{attribute 'TcRpcEnable'}
METHOD MoveModulo : itfAxisCommand
END_METHOD

{attribute 'TcRpcEnable'}
METHOD MoveRelative : itfAxisCommand
VAR_INPUT
	Distance		: REAL;
	Velocity		: REAL;
	Acceleration	: REAL;
	Deceleration	: REAL;
//	Jerk			: REAL;
//	BufferMode		: MC_BUFFER_MODE;
	Options         : Tc3_DriveMotionControl.ST_MoveOptions;
END_VAR
VAR
	itfAxisCommand   : itfAxisCommand;
	_Command         : ST_Command;
END_VAR
MC.MoveRelative(
	Axis:= Axis, 
	Execute:= TRUE, 
	Distance:= Distance, 
	Velocity:= Velocity, 
	Acceleration:= Acceleration, 
	Deceleration:= Deceleration, 
	Options:= Options, 
	Done=> _Command.Done, 
	Busy=> _Command.Busy, 
	Active=>  _Command.Active, 
	CommandAborted=>  _Command.CommandAborted, 
	Error=> _Command.Error, 
	ErrorID=> _Command.ErrorID_Udint);
	
MC.MoveRelative(
	Axis:= Axis, 
	Execute:= FALSE);		
	
itfAxisCommand.Done 				:=  _Command.Done; //AND ActualPosition = ActualPosition + Distance;             
itfAxisCommand.Busy   				:=	_Command.Busy;
itfAxisCommand.Active 				:=	_Command.Active;
itfAxisCommand.CommandAborted		:=	_Command.CommandAborted;
itfAxisCommand.Error 				:=	_Command.Error;
itfAxisCommand.ErrorID_Udint 		:=	_Command.ErrorID_Udint;

MoveRelative := itfAxisCommand;
END_METHOD

{attribute 'TcRpcEnable'}
METHOD MoveVelocity : itfContinuousAxisCommand
VAR_INPUT
	Velocity	: REAL;
	Acceleration	: REAL;
	Deceleration	: REAL;
	Jerk	: REAL;
	Direction	: MC_Direction;
	BufferMode	: MC_BUFFER_MODE;
END_VAR
END_METHOD

{attribute 'TcRpcEnable'}
METHOD Stop : itfAxisCommand
VAR_INPUT
	Deceleration	: REAL;
	Jerk	: REAL;
END_VAR
END_METHOD

{warning 'Agregar implementación de propiedad'}
PROPERTY Error : BOOL
GET
END_GET
END_PROPERTY

{warning 'Agregar implementación de propiedad'}
PROPERTY ErrorId : WORD
GET
END_GET
END_PROPERTY

{warning 'Agregar implementación de propiedad'}
PROPERTY ErrorId_Udint_Status : UDINT
GET
END_GET
END_PROPERTY

{warning 'Agregar implementación de propiedad'}
PROPERTY IsHomed : BOOL
GET
END_GET
END_PROPERTY

{warning 'Agregar implementación de propiedad'}
PROPERTY MotionStatus : MOTION_STATUS
GET
END_GET
END_PROPERTY

{warning 'Agregar implementación de propiedad'}
PROPERTY PowerOn : BOOL
GET
PowerOn := _PowerOn;
END_GET
END_PROPERTY

{warning 'Agregar implementación de propiedad'}
PROPERTY Simulation : BOOL
GET
END_GET
END_PROPERTY

PROPERTY Status : Tc3_DriveMotionControl.MC_AxisStates
GET
VAR
	AxisStates : Tc3_DriveMotionControl.MC_AxisStates;
END_VAR
//CASE Axis.Status.MotionState OF 
//    MC_AXISSTATE_UNDEFINED : 
//         AxisStates := MC_AxisStates.MC_AXISSTATE_UNDEFINED;
//	MC_AXISSTATE_DISABLED:
//		AxisStates := MC_AxisStates.MC_AXISSTATE_DISABLED;
//	MC_AXISSTATE_STANDSTILL:
//		AxisStates := MC_AxisStates.MC_AXISSTATE_STANDSTILL;
//	MC_AXISSTATE_ERRORSTOP:		
//		AxisStates := MC_AxisStates.MC_AXISSTATE_ERRORSTOP;
//	MC_AXISSTATE_STOPPING:			
//		AxisStates := MC_AxisStates.MC_AXISSTATE_STOPPING;
//	MC_AXISSTATE_HOMING:			
//		AxisStates := MC_AxisStates.MC_AXISSTATE_HOMING;
//	MC_AXISSTATE_DISCRETEMOTION:			
//		AxisStates := MC_AxisStates.MC_AXISSTATE_DISCRETEMOTION;
//	MC_AXISSTATE_CONTINOUSMOTION:			
//		AxisStates := MC_AxisStates.MC_AXISSTATE_CONTINOUSMOTION;
////	MC_AXISSTATE_SYNCHRONIZEDMOTION:			
////		AxisStates := MC_AxisStates.MC_AXISSTATE_SYNCHRONIZEDMOTION;
//END_CASE;

//Status := AxisStates;

Status := Axis.Status.MotionState;
END_GET
END_PROPERTY

{warning 'Agregar implementación de método'}
METHOD AbortTrigger : itfCommand
END_METHOD

{warning 'Agregar implementación de método'}
METHOD TouchProbe : itfCommand
END_METHOD

END_FUNCTION_BLOCK

// TwinCAT Library Template/VendorImplementation/TcAxis_Base
FUNCTION_BLOCK ABSTRACT TcAxis_Base IMPLEMENTS itfAxis_Tc3_DriveMotionControl
//VAR_INPUT
//END_VAR
//VAR_OUTPUT
//END_VAR
//VAR
//END_VAR

{warning 'Agregar implementación de propiedad'}
PROPERTY ActualPosition : REAL
GET
END_GET
END_PROPERTY

{warning 'Agregar implementación de propiedad'}
PROPERTY ActualVelocity : REAL
GET
END_GET
END_PROPERTY

{attribute 'TcRpcEnable'}
{warning 'Agregar implementación de método'}
METHOD ABSTRACT Power : itfCommand
VAR_INPUT
//	Enable	: BOOL;
//	EnablePositive	: BOOL;
//	EnableNegative	: BOOL;
END_VAR
END_METHOD

{attribute 'TcRpcEnable'}
{warning 'Agregar implementación de método'}
METHOD Reset : itfCommand
END_METHOD

{warning 'Agregar implementación de método'}
METHOD SetPosition : itfCommand
VAR_INPUT
	Position	: REAL;
	Relative	: BOOL;
	(*	ExecutionMode	: MC_ExecutionMode;*)
	ExecutionMode	: Tc2_MC2.ST_SetPositionOptions;
END_VAR
END_METHOD

{warning 'Agregar implementación de método'}
METHOD Halt : itfAxisCommand
VAR_INPUT
	Deceleration	: REAL;
	Jerk	: REAL;
	BufferMode	: MC_BUFFER_MODE;
END_VAR
END_METHOD

{warning 'Agregar implementación de método'}
METHOD Home : itfAxisCommand
VAR_INPUT
	Position	: REAL;
	Velocity	: REAL;
	EndVelocity	: REAL;
	Acceleration	: REAL;
	Deceleration	: REAL;
	Jerk	: REAL;
	Direction	: MC_Direction;
	HomingMode	: INT;
	BufferMode	: MC_BUFFER_MODE;
END_VAR
END_METHOD

{warning 'Agregar implementación de método'}
METHOD Jog : itfAxisCommand
VAR_INPUT
	JogForward	: BOOL;
	JogBackwards	: BOOL;
	Mode	: Tc2_MC2.E_JogMode;
	Position	: LREAL;
	Velocity	: LREAL;
	Acceleration	: LREAL;
	Deceleration	: LREAL;
	Jerk	: LREAL;
END_VAR
END_METHOD

{attribute 'TcRpcEnable'}
{warning 'Agregar implementación de método'}
METHOD ABSTRACT MoveAbsolute : itfAxisCommand
VAR_INPUT
//	Position	: REAL;
//	Velocity	: REAL;
//	Acceleration	: REAL;
//	Deceleration	: REAL;
//	Jerk	: REAL;
//	Direction	: MC_Direction;
//	BufferMode	: MC_BUFFER_MODE;
END_VAR
END_METHOD

{warning 'Agregar implementación de método'}
METHOD MoveModulo : itfAxisCommand
END_METHOD

{attribute 'TcRpcEnable'}
{warning 'Agregar implementación de método'}
METHOD MoveRelative : itfAxisCommand
VAR_INPUT
	Distance	: REAL;
	Velocity	: REAL;
	Acceleration	: REAL;
	Deceleration	: REAL;
	Jerk	: REAL;
	BufferMode	: MC_BUFFER_MODE;
END_VAR
END_METHOD

{warning 'Agregar implementación de método'}
METHOD MoveVelocity : itfContinuousAxisCommand
VAR_INPUT
	Velocity	: REAL;
	Acceleration	: REAL;
	Deceleration	: REAL;
	Jerk	: REAL;
	Direction	: MC_Direction;
	BufferMode	: MC_BUFFER_MODE;
END_VAR
END_METHOD

{warning 'Agregar implementación de método'}
METHOD Stop : itfAxisCommand
VAR_INPUT
	Deceleration	: REAL;
	Jerk	: REAL;
END_VAR
END_METHOD

{warning 'Agregar implementación de propiedad'}
PROPERTY Error : BOOL
GET
END_GET
END_PROPERTY

{warning 'Agregar implementación de propiedad'}
PROPERTY ErrorId : WORD
GET
END_GET
END_PROPERTY

{warning 'Agregar implementación de propiedad'}
PROPERTY ErrorId_Udint_Status : UDINT
GET
END_GET
END_PROPERTY

{warning 'Agregar implementación de propiedad'}
PROPERTY IsHomed : BOOL
GET
END_GET
END_PROPERTY

{warning 'Agregar implementación de propiedad'}
PROPERTY MotionStatus : MOTION_STATUS
GET
END_GET
END_PROPERTY

{warning 'Agregar implementación de propiedad'}
PROPERTY PowerOn : BOOL
GET
END_GET
END_PROPERTY

{warning 'Agregar implementación de propiedad'}
PROPERTY Simulation : BOOL
GET
END_GET
END_PROPERTY

PROPERTY Status : MC_AxisStates
GET
END_GET
END_PROPERTY

{warning 'Agregar implementación de método'}
METHOD AbortTrigger : itfCommand
END_METHOD

{warning 'Agregar implementación de método'}
METHOD TouchProbe : itfCommand
END_METHOD

END_FUNCTION_BLOCK

// TwinCAT Library Template/Part1Definition/Interfaces/itfAxis_Tc3_DriveMotionControl
INTERFACE itfAxis_Tc3_DriveMotionControl

{warning 'add property implementation'}
PROPERTY ActualPosition : REAL
GET
END_GET
END_PROPERTY

{warning 'add property implementation'}
PROPERTY ActualVelocity : REAL
GET
END_GET
END_PROPERTY

{attribute 'TcRpcEnable'}
//METHOD ABSTRACT Power	: itfCommand
METHOD Power	: itfCommand
VAR_INPUT
	Enable				: BOOL;
//	EnablePositive		: BOOL;
//	EnableNegative		: BOOL;
END_VAR
END_METHOD

{attribute 'TcRpcEnable'}
METHOD Reset : itfCommand
END_METHOD

{attribute 'TcRpcEnable'}
METHOD SetPosition 	: itfCommand
VAR_INPUT
	Position		: REAL;
	Relative		: BOOL;
//	ExecutionMode	: MC_ExecutionMode;
	ExecutionMode	: Tc2_MC2.ST_SetPositionOptions;
END_VAR
END_METHOD

{attribute 'TcRpcEnable'}
METHOD Halt 		: itfAxisCommand
VAR_INPUT
	Deceleration	: REAL;
	Jerk			: REAL;
	BufferMode		: MC_BUFFER_MODE;
END_VAR
END_METHOD

{attribute 'TcRpcEnable'}
METHOD Home 		: itfAxisCommand
VAR_INPUT
	Position		: REAL;
	Velocity		: REAL;
	EndVelocity		: REAL;
	Acceleration	: REAL;
	Deceleration	: REAL;
	Jerk			: REAL;
	Direction		: MC_Direction;
	HomingMode		: INT;
	BufferMode		: MC_BUFFER_MODE;
END_VAR
END_METHOD

{attribute 'TcRpcEnable'}
METHOD Jog 			: itfAxisCommand
VAR_INPUT
    JogForward 		: BOOL;
    JogBackwards 	: BOOL;
    Mode     		: Tc2_MC2.E_JogMode;
    Position        : LREAL;
    Velocity        : LREAL;
    Acceleration 	: LREAL;
    Deceleration 	: LREAL;
    Jerk     		: LREAL;
END_VAR
END_METHOD

{attribute 'TcRpcEnable'}
METHOD MoveAbsolute : itfAxisCommand
//METHOD ABSTRACT MoveAbsolute : itfAxisCommand
VAR_INPUT
	Position		: REAL;
	Velocity		: REAL;
	Acceleration	: REAL;
	Deceleration	: REAL;
//	Jerk			: REAL;
//	Direction		: MC_Direction;
//	BufferMode		: MC_BUFFER_MODE;
	Options         : Tc3_DriveMotionControl.ST_MoveOptions;
END_VAR
END_METHOD

{attribute 'TcRpcEnable'}
METHOD MoveModulo : itfAxisCommand
VAR_INPUT
END_VAR
END_METHOD

{attribute 'TcRpcEnable'}
METHOD MoveRelative : itfAxisCommand
VAR_INPUT
	Distance		: REAL;
	Velocity		: REAL;
	Acceleration	: REAL;
	Deceleration	: REAL;
//	Jerk			: REAL;
//	BufferMode		: MC_BUFFER_MODE;
	Options         : Tc3_DriveMotionControl.ST_MoveOptions;
END_VAR
END_METHOD

{attribute 'TcRpcEnable'}
METHOD MoveVelocity : itfContinuousAxisCommand
VAR_INPUT
	Velocity		: REAL;
	Acceleration	: REAL;
	Deceleration	: REAL;
	Jerk			: REAL;
	Direction		: MC_Direction;
	BufferMode		: MC_BUFFER_MODE;
END_VAR
END_METHOD

{attribute 'TcRpcEnable'}
METHOD Stop 		: itfAxisCommand
VAR_INPUT
	Deceleration	: REAL;
	Jerk			: REAL;
END_VAR
END_METHOD

PROPERTY Error : BOOL
GET
END_GET
END_PROPERTY

{warning 'add property implementation'}
PROPERTY ErrorId : WORD
GET
END_GET
END_PROPERTY

PROPERTY ErrorId_Udint_Status : UDINT
GET
END_GET
END_PROPERTY


PROPERTY IsHomed : BOOL
GET
END_GET
END_PROPERTY

{warning 'add property implementation'}
PROPERTY MotionStatus : MOTION_STATUS
GET
END_GET
END_PROPERTY

{attribute ‘monitoring’ := ‘call’}
PROPERTY PowerOn : BOOL
GET
END_GET
END_PROPERTY

{warning 'add property implementation'}
PROPERTY Simulation : BOOL
GET
END_GET
END_PROPERTY

PROPERTY Status : Tc3_DriveMotionControl.MC_AxisStates
GET
END_GET
END_PROPERTY

METHOD AbortTrigger : itfCommand
VAR_INPUT
END_VAR
END_METHOD

METHOD TouchProbe : itfCommand
VAR_INPUT
END_VAR
END_METHOD

END_INTERFACE

// Examples/_MAIN_Examples
PROGRAM _MAIN_Examples
VAR
//	fbAxis_X1 				: TcAxis_Tc2_MC2;
			
//	fbSum : FB_Sum;
END_VAR

//Examples Tc2_MC2:
WareHousingExample_Tc2_MC2();
//LabelingExample();
//CamGearExample();

//Examples Tc3_DriveMotionControl:
WareHousingExample_Tc3_DriveMotionControl();

END_PROGRAM

// Examples/LabelingExample
PROGRAM LabelingExample
VAR
	AXIS_REF_LabelDrive			: TC2_MC2.AXIS_REF;
	AXIS_REF_Conveyor 			: TC2_MC2.AXIS_REF;

	// Hardware definitions
	LabelDrive 			: TcAxis_Tc2_MC2;
	Conveyor 			: TcAxis_Tc2_MC2;
	LabelLength 		: REAL := 100;
	SensorDistance 		: REAL := 10;
	Velocity 			: REAL := 5;
	ProductDetection 	: BOOL := FALSE;
	DelayTimer 			: TON;
	
	// States
	ConveyorState 		: INT := 0;
	LabelDriveState 	: INT := 0;
	
	// Control
	Start 				: BOOL := FALSE;
	
	// Commands
	ConveyorMove 		: itfCommand;
	LabelDriveMove 		: itfCommand;
END_VAR


LabelDrive(Axis:= AXIS_REF_LabelDrive);
Conveyor(Axis:= AXIS_REF_Conveyor);

// Run the timer. As it is a classic FB it should be called every cycle
DelayTimer(IN:=ProductDetection, PT:= INT_TO_TIME(REAL_TO_INT(SensorDistance * 1000 / Velocity)));

CASE ConveyorState OF
	0: // Disabled
		IF Start THEN
			ConveyorState := ConveyorState + 1;
		END_IF
		
	1: // Power On
		Conveyor.Power(Enable:=TRUE, EnablePositive:=TRUE, EnableNegative:=TRUE);
		//IF Conveyor.Status = AXIS_STATUS.Standstill THEN
	  IF Conveyor.Status = Tc2_MC2.MC_AXISSTATE_STANDSTILL THEN
			ConveyorState := ConveyorState + 1;
		END_IF
		
	2: // Wait for LabelDrive 
		//IF LabelDrive.Status = AXIS_STATUS.Standstill THEN
		IF LabelDrive.Status =  Tc2_MC2.MC_AXISSTATE_STANDSTILL THEN
			ConveyorMove := Conveyor.MoveVelocity(Velocity:=Velocity, Acceleration:=0, Deceleration:=0, Jerk:=0, Direction:=MC_Direction.mcPositiveDirection, BufferMode:=MC_BUFFER_MODE.mcAborting);
			ConveyorState := ConveyorState + 1;
		END_IF
		
	3: // Moving
		IF NOT Start THEN
			ConveyorMove := Conveyor.Halt(Deceleration:=0, Jerk:=0, BufferMode:=MC_BUFFER_MODE.mcAborting);
			ConveyorState := ConveyorState + 1;
		END_IF
		
	4: // Stopping
		IF ConveyorMove.Done THEN
			ConveyorState := ConveyorState + 1;
		END_IF
		
	5: // Power off
		Conveyor.Power(Enable:=FALSE, EnablePositive:=FALSE, EnableNegative:=FALSE);
		IF Conveyor.Status = AXIS_STATUS.Disabled THEN
			ConveyorState := 0;
		END_IF
END_CASE

CASE LabelDriveState OF
	0: // Disabled
		IF Start THEN
			LabelDriveState := LabelDriveState + 1;
		END_IF
		
	1: // Power On
		LabelDrive.Power(Enable:=TRUE, EnablePositive:=TRUE, EnableNegative:=TRUE);
		//IF LabelDrive.Status = AXIS_STATUS.Standstill THEN
		IF LabelDrive.Status = Tc2_MC2.MC_AXISSTATE_STANDSTILL THEN
			LabelDriveState := LabelDriveState + 1;
		END_IF
		
	2: // Wait for Conveyor 
		//IF Conveyor.Status = AXIS_STATUS.Standstill THEN
		IF Conveyor.Status = Tc2_MC2.MC_AXISSTATE_STANDSTILL THEN
			LabelDriveState := LabelDriveState + 1;
		END_IF
						
	3: // Wait for product
		IF NOT Start THEN
			LabelDriveState := 5;
		END_IF
		IF DelayTimer.Q THEN
			LabelDriveMove := LabelDrive.MoveRelative(Distance:=LabelLength, Velocity:=Velocity, Acceleration:=0, Deceleration:=0, Jerk:=0, BufferMode:=MC_BUFFER_MODE.mcAborting);
			LabelDriveState := LabelDriveState + 1;
		END_IF
		
	4: // Wait for label to be transfered
		IF LabelDriveMove.Done AND NOT DelayTimer.Q THEN
			LabelDriveState := 3;
		END_IF
		
	5: // Power off
		Conveyor.Power(Enable:=FALSE, EnablePositive:=FALSE, EnableNegative:=FALSE);
		IF Conveyor.Status = AXIS_STATUS.Disabled THEN
			LabelDriveState := 0;
		END_IF
	
END_CASE

END_PROGRAM

// Examples/CamGearExample
PROGRAM CamGearExample
VAR
	// Hardware definitions
	TcMasterDrive 	: TcAxis_Tc2_MC2;
	TcCamDrive 		: TcAxis_Tc2_MC2;
	TcGearDrive 	: TcAxis_Tc2_MC2;
	
	
	MasterDrive 	: itfAxis_Tc2_MC2;
	CamDrive 		: itfAxis_Tc2_MC2;
	GearDrive 		: itfAxis_Tc2_MC2;
	Table 			: TcCamTable;
	TableData 		: MC_CAM_REF;
	Velocity 		: REAL := 5;
	
	// States
	MasterState 	: INT := 0;
	CamState 		: INT := 0;
	GearState 		: INT := 0;
	
	// Control
	Start 			: BOOL := FALSE;
	
	// Commands
	MasterMove 		: itfCommand;
	TableSet 		: itfCommand;
	CamMove 		: itfSynchronizedAxisCommand;
	GearMove 		: itfSynchronizedAxisCommand;
END_VAR


MasterDrive:= TcMasterDrive;
CamDrive := TcCamDrive;
GearDrive := TcGearDrive;

CASE MasterState OF
	0: // Disabled
		IF Start THEN
			MasterState := MasterState + 1;
		END_IF
		
	1: // Power On
		MasterDrive.Power(Enable:=TRUE, EnablePositive:=TRUE, EnableNegative:=TRUE);
		IF MasterDrive.Status = AXIS_STATUS.Standstill THEN
			MasterState := MasterState + 1;
		END_IF
		
	2: // Wait for other drives 
		IF CamMove.InSync AND GearMove.InSync THEN
			MasterMove := MasterDrive.MoveVelocity(Velocity:=Velocity, Acceleration:=0, Deceleration:=0, Jerk:=0, Direction:=MC_Direction.mcPositiveDirection, BufferMode:=MC_BUFFER_MODE.mcAborting);
			MasterState := MasterState + 1;
		END_IF
		
	3: // Moving
		IF NOT Start THEN
			MasterMove:= MasterDrive.Halt(Deceleration:=0, Jerk:=0, BufferMode:=MC_BUFFER_MODE.mcAborting);
			MasterState := MasterState + 1;
		END_IF
		
	4: // Stopping
		IF NOT MasterMove.Done THEN
			MasterState := MasterState + 1;
		END_IF
		
	5: // Power off
		MasterDrive.Power(Enable:=FALSE, EnablePositive:=FALSE, EnableNegative:=FALSE);
		IF MasterDrive.Status = AXIS_STATUS.Disabled THEN
			MasterState := 0;
		END_IF
END_CASE

CASE CamState OF
	0: // Disabled
		IF Start THEN
			CamState := CamState + 1;
		END_IF
		
	1: // Power On
		CamDrive.Power(Enable:=TRUE, EnablePositive:=TRUE, EnableNegative:=TRUE);
		IF CamDrive.Status = AXIS_STATUS.Standstill AND MasterDrive.Status = AXIS_STATUS.Standstill THEN
			TableSet := Table.Select(CamTable:=TableData, Periodic:=TRUE, MasterAbsolute:=TRUE, SlaveAbsolute:=TRUE);
			CamState := CamState + 1;
		END_IF
		
	2: // Set CAM Table
		IF TableSet.Done THEN
			CamMove := CamDrive.CamIn(Master:=MasterDrive, MasterOffset:=0, SlaveOffset:=0, MasterScaling:=1, SlaveScaling:=1, MasterStartDistance:=0, MasterSyncPosition:=0, 
				StartMode:=MC_StartMode.mcRelative, MasterValueSource:=MC_Source.mcSetValue,CamTable:=Table, BufferMode:=MC_BUFFER_MODE.mcAborting);
			CamState := CamState + 1;
		END_IF
		
	3: // Synchronized
		IF NOT Start THEN
			CamDrive.Release();
			CamState := CamState + 1;
		END_IF
		
	4: // Power off
		CamDrive.Power(Enable:=FALSE, EnablePositive:=FALSE, EnableNegative:=FALSE);
		IF CamDrive.Status = AXIS_STATUS.Disabled THEN
			CamState := 0;
		END_IF
END_CASE

CASE GearState OF
	0: // Disabled
		IF Start THEN
			GearState := GearState + 1;
		END_IF
		
	1: // Power On
		GearDrive.Power(Enable:=TRUE, EnablePositive:=TRUE, EnableNegative:=TRUE);
		IF GearDrive.Status = AXIS_STATUS.Standstill AND MasterDrive.Status = AXIS_STATUS.Standstill THEN
			GearMove := GearDrive.GearIn(Master:=MasterDrive, Ratio:=2, MasterValueSource:=MC_Source.mcSetValue,Acceleration:=0, Deceleration:=0, Jerk:=0, BufferMode:=MC_BUFFER_MODE.mcAborting);
			GearState := GearState + 1;
		END_IF
		
	2: // Synchronized
		IF NOT Start THEN
			GearDrive.Release();
			GearState := GearState + 1;
		END_IF
		
	3: // Power off
		GearDrive.Power(Enable:=FALSE, EnablePositive:=FALSE, EnableNegative:=FALSE);
		IF GearDrive.Status = AXIS_STATUS.Disabled THEN
			GearState := 0;
		END_IF
END_CASE

END_PROGRAM

// TwinCAT Library Template/VendorImplementation/TcCamTable
FUNCTION_BLOCK TcCamTable IMPLEMENTS itfCamTable
VAR_INPUT
END_VAR
VAR_OUTPUT
END_VAR
VAR
END_VAR

{warning 'add method implementation '}
METHOD Select 		: itfCommand
VAR_INPUT	
	Periodic		: BOOL;
	MasterAbsolute	: BOOL;
	SlaveAbsolute	: BOOL;
	CamTable		: MC_CAM_REF;
END_VAR
VAR
	
END_VAR
END_METHOD

END_FUNCTION_BLOCK

// Project Information/F_GetCompany
// This function has been automatically generated from the project information.
{attribute 'signature_flag' := '1073741824'}
{attribute 'TcGenerated'}
{attribute 'no-analysis'}
FUNCTION F_GetCompany : WSTRING
VAR_INPUT
	
END_VAR

F_GetCompany := "TcMotion";

END_FUNCTION

// Project Information/F_GetTitle
// This function has been automatically generated from the project information.
{attribute 'signature_flag' := '1073741824'}
{attribute 'TcGenerated'}
{attribute 'no-analysis'}
FUNCTION F_GetTitle : WSTRING
VAR_INPUT
	
END_VAR

F_GetTitle := "TcMotion_Component";

END_FUNCTION

// Project Information/F_GetVersion
// This function has been automatically generated from the project information.
{attribute 'signature_flag' := '1073741824'}
{attribute 'TcGenerated'}
{attribute 'no-analysis'}
FUNCTION F_GetVersion : ST_LibVersion
VAR_INPUT
	
END_VAR

F_GetVersion.iMajor := 1;
F_GetVersion.iMinor := 0;
F_GetVersion.iBuild := 0;
F_GetVersion.iRevision := 8;
F_GetVersion.sVersion := '1.0.0.8';
F_GetVersion.nFlags := 0;

END_FUNCTION

// TwinCAT Library Template/Part1Definition/Interfaces/itfAxis_Tc2_MC2_Camming
INTERFACE itfAxis_Tc2_MC2_Camming

(*
!!!! It would have to be another library with this new extension for the Axis, because if not in TwinCAT this new license is added:
!!!! TF5050 TC3 NC Camming !!!!!!*)

{attribute 'TcRpcEnable'}
METHOD CamIn 			: itfSynchronizedAxisCommand
VAR_INPUT
//	Master				: itfAxis;
	Master				: Tc2_MC2.AXIS_REF;
	Slave				: Tc2_MC2.AXIS_REF;	
	MasterOffset		: REAL;
	SlaveOffset			: REAL;
	MasterScaling		: REAL;
	SlaveScaling		: REAL;
	MasterStartDistance	: REAL;
	MasterSyncPosition	: REAL;
	StartMode			: MC_StartMode;
	MasterValueSource	: MC_Source;
//	CamTable			: itfCamTable;
	CamTableID			: Tc2_MC2_Camming.MC_CAM_ID;
	BufferMode			: MC_BUFFER_MODE;
END_VAR
END_METHOD

{attribute 'TcRpcEnable'}
METHOD CamOut : : itfSynchronizedAxisCommand
VAR_INPUT
END_VAR
END_METHOD

{attribute 'TcRpcEnable'}
METHOD CamScaling : itfSynchronizedAxisCommand
VAR_INPUT
END_VAR
END_METHOD

{attribute 'TcRpcEnable'}
METHOD CamTableSelect  : itfSynchronizedAxisCommand
VAR_INPUT
END_VAR
END_METHOD

{attribute 'TcRpcEnable'}
METHOD ReadMotionFunction : itfSynchronizedAxisCommand
VAR_INPUT
END_VAR
END_METHOD

{attribute 'TcRpcEnable'}
METHOD ReadMotionFunctionPoint : itfSynchronizedAxisCommand
VAR_INPUT
END_VAR
END_METHOD

{attribute 'TcRpcEnable'}
METHOD ReadMotionFunctionValues : itfSynchronizedAxisCommand
VAR_INPUT
END_VAR
END_METHOD

{attribute 'TcRpcEnable'}
METHOD SetCamOnlineChangeMode : itfSynchronizedAxisCommand
VAR_INPUT
END_VAR
END_METHOD

{attribute 'TcRpcEnable'}
METHOD WriteMotionFunction : itfSynchronizedAxisCommand
VAR_INPUT
END_VAR
END_METHOD

{attribute 'TcRpcEnable'}
METHOD WriteMotionFunctionPoint : itfSynchronizedAxisCommand
VAR_INPUT
END_VAR
END_METHOD

{attribute 'TcRpcEnable'}
METHOD CamAdd : itfSynchronizedAxisCommand
VAR_INPUT
END_VAR
END_METHOD

{attribute 'TcRpcEnable'}
METHOD CamExchange : itfSynchronizedAxisCommand
VAR_INPUT
END_VAR
END_METHOD

{attribute 'TcRpcEnable'}
METHOD CamIn_V2 : itfSynchronizedAxisCommand
VAR_INPUT
END_VAR
END_METHOD

{attribute 'TcRpcEnable'}
METHOD CamRemove : itfSynchronizedAxisCommand
VAR_INPUT
END_VAR
END_METHOD

{attribute 'TcRpcEnable'}
METHOD CamScaling_V2 : itfSynchronizedAxisCommand
VAR_INPUT
END_VAR
END_METHOD

{attribute 'TcRpcEnable'}
METHOD CamInfo : itfSynchronizedAxisCommand
VAR_INPUT
END_VAR
END_METHOD

{attribute 'TcRpcEnable'}
METHOD CamInfo_V2 : itfSynchronizedAxisCommand
VAR_INPUT
END_VAR
END_METHOD

{attribute 'TcRpcEnable'}
METHOD ReadCamTableCharacteristics : itfSynchronizedAxisCommand
VAR_INPUT
END_VAR
END_METHOD

{attribute 'TcRpcEnable'}
METHOD ReadCamTableMasterPosition : itfSynchronizedAxisCommand
VAR_INPUT
END_VAR
END_METHOD

{attribute 'TcRpcEnable'}
METHOD ReadCamTableSlaveDynamics : itfSynchronizedAxisCommand
VAR_INPUT
END_VAR
END_METHOD

END_INTERFACE

// TwinCAT Library Template/Part1Definition/Interfaces/itfAxis_Tc2_MC2_FlyingSaw
INTERFACE itfAxis_Tc2_MC2_FlyingSaw

(*
!!!! It would have to be another library with this new extension for the Axis, because if not in TwinCAT this new license is added:
!!!! TF5055 TC3 NC Flying Saw !!!!!!*)

{attribute 'TcRpcEnable'}
METHOD GearInPos 		: itfSynchronizedAxisCommand
VAR_INPUT
//	Master				: itfAxis;
	Master				: Tc2_MC2.AXIS_REF;
	Slave				: Tc2_MC2.AXIS_REF;			
	RatioNumerator		: REAL;
	RatioDenominator	: REAL;
	MasterValueSource	: MC_SOURCE;
	MasterSyncPosition	: REAL;
	SlaveSyncPosition	: REAL;
	SyncMode			: MC_SYNC_MODE;
	MasterStartDistance	: REAL;
	Velocity			: REAL;
	Acceleration		: REAL;
	Deceleration		: REAL;
	Jerk				: REAL;
	BufferMode			: MC_BUFFER_MODE;
END_VAR
END_METHOD

{attribute 'TcRpcEnable'}
METHOD GearInVelo 		: itfSynchronizedAxisCommand
VAR_INPUT
//	Master				: itfAxis;
	Master				: Tc2_MC2.AXIS_REF;
	Slave				: Tc2_MC2.AXIS_REF;			
	RatioNumerator		: REAL;
	RatioDenominator	: REAL;
	MasterValueSource	: MC_SOURCE;
	MasterSyncPosition	: REAL;
	SlaveSyncPosition	: REAL;
	SyncMode			: MC_SYNC_MODE;
	MasterStartDistance	: REAL;
	Velocity			: REAL;
	Acceleration		: REAL;
	Deceleration		: REAL;
	Jerk				: REAL;
	BufferMode			: MC_BUFFER_MODE;
END_VAR
END_METHOD

{attribute 'TcRpcEnable'}
METHOD ReadFlyingSawCharacteristics : itfSynchronizedAxisCommand
VAR_INPUT
END_VAR
END_METHOD

END_INTERFACE

// TwinCAT Library Template/VendorImplementation/TcAxis_Tc2_MC2_Camming
FUNCTION_BLOCK TcAxis_Tc2_MC2_Camming EXTENDS TcAxis_Tc2_MC2 IMPLEMENTS itfAxis_Tc2_MC2_Camming
VAR_INPUT
END_VAR
VAR_OUTPUT
END_VAR
VAR
END_VAR

{error 'Agregar implementación de método o eliminar método para utilizar la implementación básica.'}
(*
!!!! It would have to be another library with this new extension for the Axis, because if not in TwinCAT this new license is added:
!!!! TF5050 TC3 NC Camming !!!!!!*)
METHOD CamIn : itfSynchronizedAxisCommand
VAR_INPUT
	(*	Master				: itfAxis;*)
	Master	: Tc2_MC2.AXIS_REF;
	Slave	: Tc2_MC2.AXIS_REF;
	MasterOffset	: REAL;
	SlaveOffset	: REAL;
	MasterScaling	: REAL;
	SlaveScaling	: REAL;
	MasterStartDistance	: REAL;
	MasterSyncPosition	: REAL;
	StartMode	: MC_StartMode;
	MasterValueSource	: MC_Source;
	(*	CamTable			: itfCamTable;*)
	CamTableID	: Tc2_MC2_Camming.MC_CAM_ID;
	BufferMode	: MC_BUFFER_MODE;
END_VAR

VAR
	fbCamIn			 	: Tc2_MC2_Camming.MC_CamIn;	
END_VAR
(*
!!!! It would have to be another library with this new extension for the Axis, because if not in TwinCAT this new license is added:
!!!! TF5050 TC3 NC Camming !!!!!!*)

fbCamIn(
	Master:= Master, 
	Slave:= Slave, 
	Execute:= TRUE, 
	MasterOffset:= MasterOffset, 
	SlaveOffset:= SlaveOffset, 
	MasterScaling:= MasterScaling, 
	SlaveScaling:= SlaveScaling, 
	StartMode:= StartMode, 
	CamTableID:= CamTableID, //CamTable, 
	BufferMode:= , //BufferMode, 
	Options:= , 
	InSync=> , 
	Busy=> , 
	Active=> , 
	CommandAborted=> , 
	Error=> , 
	ErrorID=> );

count_delete  := count_delete + 1;
END_METHOD

END_FUNCTION_BLOCK

// TwinCAT Library Template/VendorImplementation/TcAxis_Tc2_MC2_FlyingSaw
FUNCTION_BLOCK TcAxis_Tc2_MC2_FlyingSaw EXTENDS TcAxis_Tc2_MC2 IMPLEMENTS itfAxis_Tc2_MC2_FlyingSaw
VAR_INPUT
END_VAR
VAR_OUTPUT
END_VAR
VAR
END_VAR

{error 'Agregar implementación de método o eliminar método para utilizar la implementación básica.'}
(*
!!!! It would have to be another library with this new extension for the Axis, because if not in TwinCAT this new license is added:
!!!! TF5055 TC3 NC Flying Saw !!!!!!*)
METHOD GearInPos : itfSynchronizedAxisCommand
VAR_INPUT
	(*	Master				: itfAxis;*)
	Master	: Tc2_MC2.AXIS_REF;
	Slave	: Tc2_MC2.AXIS_REF;
	RatioNumerator	: REAL;
	RatioDenominator	: REAL;
	MasterValueSource	: MC_SOURCE;
	MasterSyncPosition	: REAL;
	SlaveSyncPosition	: REAL;
	SyncMode	: MC_SYNC_MODE;
	MasterStartDistance	: REAL;
	Velocity	: REAL;
	Acceleration	: REAL;
	Deceleration	: REAL;
	Jerk	: REAL;
	BufferMode	: MC_BUFFER_MODE;
END_VAR

VAR
	fbGearInPos			: Tc2_MC2_FlyingSaw.MC_GearInPos;	
END_VAR
(*
!!!! It would have to be another library with this new extension for the Axis, because if not in TwinCAT this new license is added:
!!!! TF5055 TC3 NC Flying Saw !!!!!!*)

fbGearInPos(
	Master:= Master, 
	Slave:= Slave, 
	Execute:= , 
	RatioNumerator:= , 
	RatioDenominator:= , 
	MasterSyncPosition:= , 
	SlaveSyncPosition:= , 
	SyncMode:= , 
	MasterStartDistance:= , 
	Velocity:= , 
	Acceleration:= , 
	Deceleration:= , 
	Jerk:= , 
	BufferMode:= , 
	Options:= , 
	StartSync=> , 
	InSync=> , 
	Busy=> , 
	Active=> , 
	CommandAborted=> , 
	Error=> , 
	ErrorID=> );


count_delete  := count_delete + 1;
END_METHOD

END_FUNCTION_BLOCK

// TwinCAT Library Template/VendorImplementation/TcContinuousAxisCommand
FUNCTION_BLOCK TcContinuousAxisCommand IMPLEMENTS itfContinuousAxisCommand
VAR_INPUT
END_VAR
VAR_OUTPUT
END_VAR
VAR
END_VAR

{warning 'add method implementation '}
METHOD Abort : MC_Error
END_METHOD

{warning 'add property implementation'}
PROPERTY Active : BOOL
GET
END_GET
END_PROPERTY

{warning 'add property implementation'}
PROPERTY Busy : BOOL
GET
END_GET
END_PROPERTY

{warning 'add property implementation'}
PROPERTY Command : MC_COMMAND_REF
GET
END_GET
END_PROPERTY

{warning 'add property implementation'}
PROPERTY CommandAborted : BOOL
GET
END_GET
END_PROPERTY

{warning 'add property implementation'}
PROPERTY Done : BOOL
GET
END_GET
END_PROPERTY

{warning 'add property implementation'}
PROPERTY Error : BOOL
GET
END_GET
END_PROPERTY

{warning 'add property implementation'}
PROPERTY ErrorId : MC_Error
GET
END_GET
END_PROPERTY

{warning 'add property implementation'}
PROPERTY InVelocity : BOOL
GET
END_GET
END_PROPERTY

{warning 'add method implementation '}
METHOD Update 		: MC_Error
VAR_INPUT
	Position		: REAL;
	Velocity		: REAL;
	EndVelocity		: REAL;
	Acceleration	: REAL;
	Deceleration	: REAL;
	Jerk			: REAL;
END_VAR
END_METHOD

{warning 'add method implementation '}
METHOD Wait 		: MC_Error (* This method only makes sense in the IEC 61499 environment*)
VAR_INPUT
	Timeout			: TIME;
	AbortOnTimeout	: BOOL;
END_VAR
END_METHOD

END_FUNCTION_BLOCK

// TwinCAT Library Template/VendorImplementation/TcSynchronizedAxisCommand
FUNCTION_BLOCK TcSynchronizedAxisCommand IMPLEMENTS itfSynchronizedAxisCommand
VAR_INPUT
END_VAR
VAR_OUTPUT
END_VAR
VAR
END_VAR

{warning 'add method implementation '}
METHOD Abort : MC_Error
END_METHOD

{warning 'add property implementation'}
PROPERTY Active : BOOL
GET
END_GET
END_PROPERTY

{warning 'add property implementation'}
PROPERTY Busy : BOOL
GET
END_GET
END_PROPERTY

{warning 'add property implementation'}
PROPERTY Command : MC_COMMAND_REF
GET
END_GET
END_PROPERTY

{warning 'add property implementation'}
PROPERTY CommandAborted : BOOL
GET
END_GET
END_PROPERTY

{warning 'add property implementation'}
PROPERTY Done : BOOL
GET
END_GET
END_PROPERTY

{warning 'add property implementation'}
PROPERTY Error : BOOL
GET
END_GET
END_PROPERTY

{warning 'add property implementation'}
PROPERTY ErrorId : MC_Error
GET
END_GET
END_PROPERTY

{warning 'add property implementation'}
PROPERTY InSync : BOOL
GET
Insync:= Geared;
END_GET
END_PROPERTY

{warning 'add method implementation '}
METHOD Update 		: MC_Error
VAR_INPUT
	Position		: REAL;
	Velocity		: REAL;
	EndVelocity		: REAL;
	Acceleration	: REAL;
	Deceleration	: REAL;
	Jerk			: REAL;
END_VAR
END_METHOD

{warning 'add method implementation '}
METHOD Wait 		: MC_Error (* This method only makes sense in the IEC 61499 environment*)
VAR_INPUT
	Timeout			: TIME;
	AbortOnTimeout	: BOOL;
END_VAR
END_METHOD

END_FUNCTION_BLOCK
